Omron CX-Programmer project 新工程 (CX-Programmer 9.73)

# PLC 新PLC1: C200HE CPU42

## Program 新程序1 (no task)
; [项目]：本项目是为“台湾大拉无板”自动化拉丝生产线设计的控制系统，通过PLC实现生产线的自动化管理。系统包含启动、错误处理、定时管理、事件计数和设备驱动模块，确保拉丝作业的正常运行。 / [设备信息]：系统涉及的物理设备包括启动按钮、停止按钮、模式选择按钮、传感器、拉丝机电机和阀门。 / [系统执行]：系统通过启动按钮启动生产线，操作员按下按钮后，程序检查异常传感器1至10是否正常。 / 若无异常且延时定时器2未超时，置位运行模式标志，此时生产线进入运行状态。 / 特别地，运行模式标志只有在启动按钮按下后才会置位，避免未触发启动时生产线意外运行。 / 运行时，电机控制1至10驱动拉丝机运转，其中电机控制1的激活必须在运行模式标志置位时才能发生，防止模式未启用时设备误动作。 / 当系统正常运行时，若检测到特定条件，激活电机控制1以驱动设备。 / 启动时，异常传感器1至10检查是否正常；运行中，若任一传感器检测到异常，则置位相应标志。 / 若延时定时器1超时，置位错误状态标志；随后通过停止控制信号停止生产线，并激活阀门2发出警报。 / 错误状态标志置位后，激活阀门2发出警报，并通过停止控制信号停止生产线。 / 延时定时器1超时置位错误状态标志；延时定时器2超时（设定为20个时间单位）后，也触发类似逻辑。 / 操作员可通过手动按钮1和手动按钮2手动控制阀门1和阀门2（如调节润滑液或冷却液），这些操作的计数记录在次数记录区中。 / 当计数达到4时，系统自动复位阀门状态，确保手动操作不会无限制累积。 / 事件计数器1记录拉丝次数，限值为3次；若达到限值，后续逻辑触发警报。 / 模式选择按钮1至9允许切换拉丝模式（如高速或低速模式），当前模式存储在模式记录区中，影响拉丝参数。 / 参数存储区保存运行数据和历史记录，便于维护和故障排查。 / 按下停止按钮后，系统置位停止控制信号以停止生产线。

### Section 段1

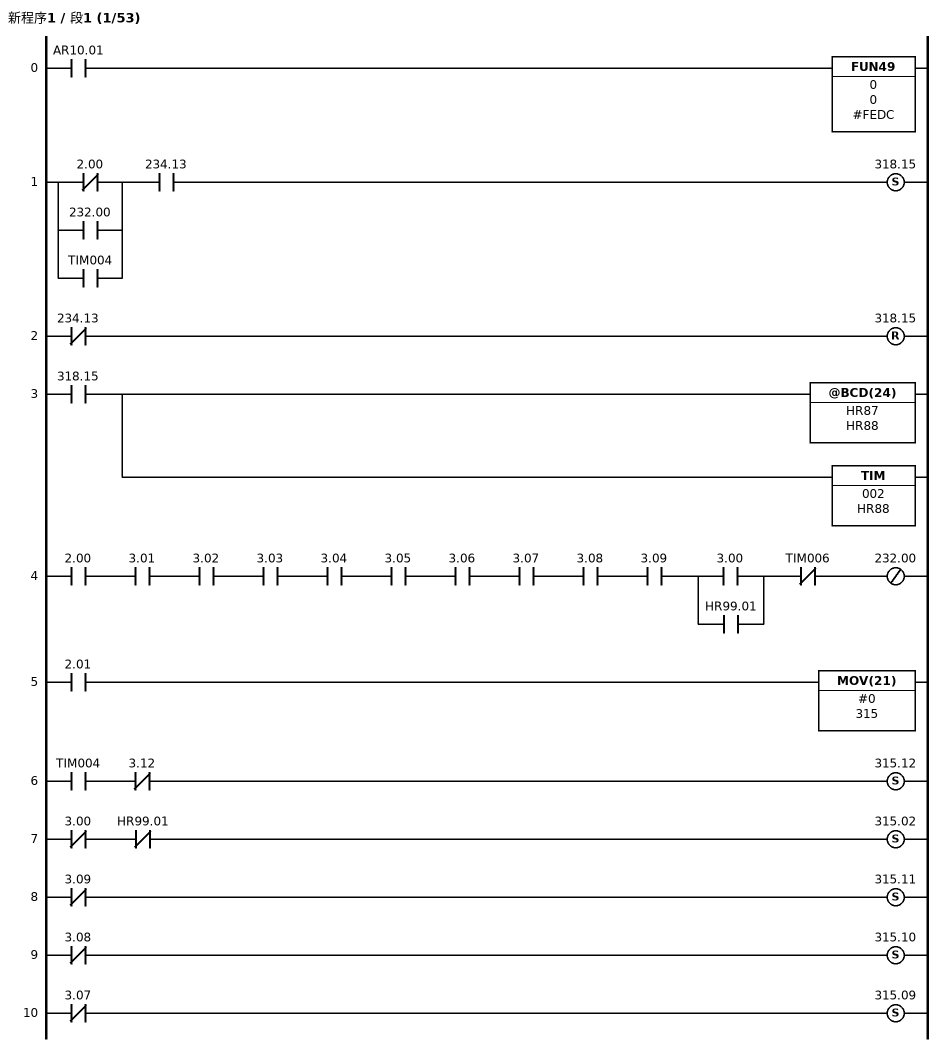
; rung 0
LD AR10.01
FUN49 0 0 #FEDC
; rung 1
LDNOT 2.00
OR 232.00
OR TIM004
AND 234.13
SET 318.15
; rung 2
LDNOT 234.13
RSET 318.15
; rung 3
LD 318.15
@BCD(24) HR87 HR88
TIM 002 HR88
; rung 4
LD 2.00
AND 3.01
AND 3.02
AND 3.03
AND 3.04
AND 3.05
AND 3.06
AND 3.07
AND 3.08
AND 3.09
LD 3.00
OR HR99.01
ANDLD
ANDNOT TIM006
OUTNOT 232.00
; rung 5
LD 2.01
MOV(21) #0 315
; rung 6
LD TIM004
ANDNOT 3.12
SET 315.12
; rung 7
LDNOT 3.00
ANDNOT HR99.01
SET 315.02
; rung 8
LDNOT 3.09
SET 315.11
; rung 9
LDNOT 3.08
SET 315.10
; rung 10
LDNOT 3.07
SET 315.09

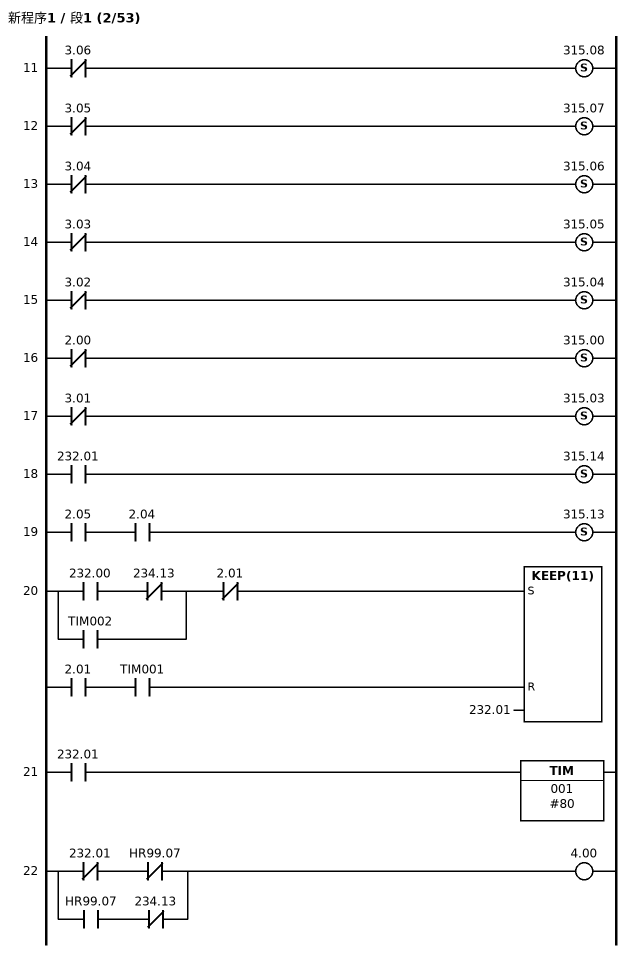
; rung 11
LDNOT 3.06
SET 315.08
; rung 12
LDNOT 3.05
SET 315.07
; rung 13
LDNOT 3.04
SET 315.06
; rung 14
LDNOT 3.03
SET 315.05
; rung 15
LDNOT 3.02
SET 315.04
; rung 16
LDNOT 2.00
SET 315.00
; rung 17
LDNOT 3.01
SET 315.03
; rung 18
LD 232.01
SET 315.14
; rung 19
LD 2.05
AND 2.04
SET 315.13
; rung 20
LD 232.00
ANDNOT 234.13
OR TIM002
ANDNOT 2.01
LD 2.01
AND TIM001
KEEP(11) 232.01
; rung 21
LD 232.01
TIM 001 #80
; rung 22
LDNOT 232.01
ANDNOT HR99.07
LD HR99.07
ANDNOT 234.13
ORLD
OUT 4.00

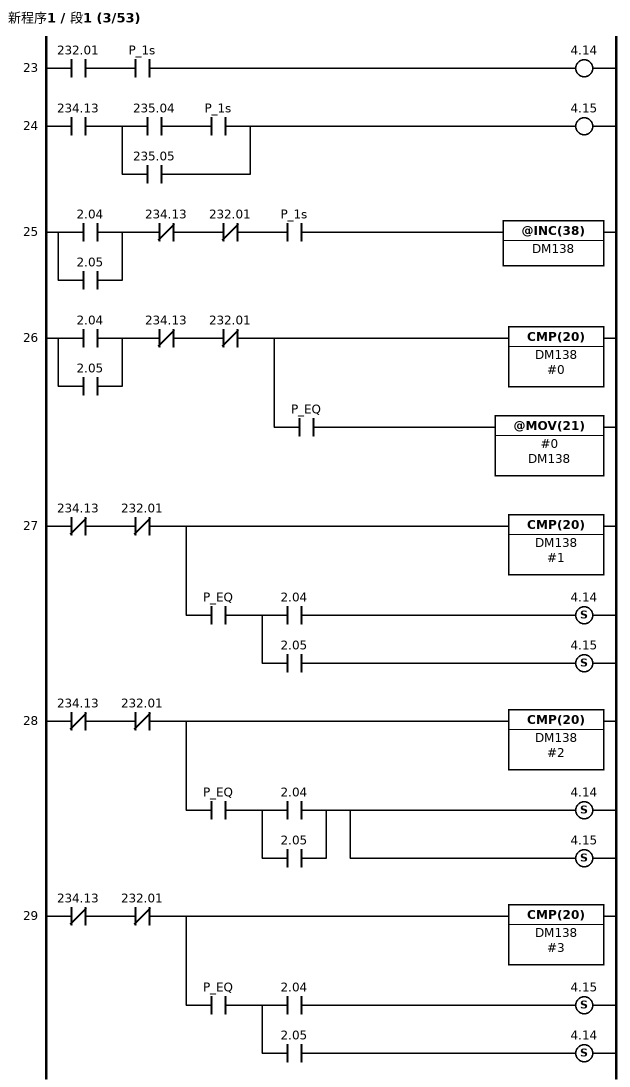
; rung 23
LD 232.01
AND P_1s
OUT 4.14
; rung 24
LD 234.13
LD 235.04
AND P_1s
OR 235.05
ANDLD
OUT 4.15
; rung 25
LD 2.04
OR 2.05
ANDNOT 234.13
ANDNOT 232.01
AND P_1s
@INC(38) DM138
; rung 26
LD 2.04
OR 2.05
ANDNOT 234.13
ANDNOT 232.01
CMP(20) DM138 #0
AND P_EQ
@MOV(21) #0 DM138
; rung 27
LDNOT 234.13
ANDNOT 232.01
CMP(20) DM138 #1
AND P_EQ
OUT TR0
AND 2.04
SET 4.14
LD TR0
AND 2.05
SET 4.15
; rung 28
LDNOT 234.13
ANDNOT 232.01
CMP(20) DM138 #2
AND P_EQ
LD 2.04
OR 2.05
ANDLD
SET 4.14
SET 4.15
; rung 29
LDNOT 234.13
ANDNOT 232.01
CMP(20) DM138 #3
AND P_EQ
OUT TR0
AND 2.04
SET 4.15
LD TR0
AND 2.05
SET 4.14

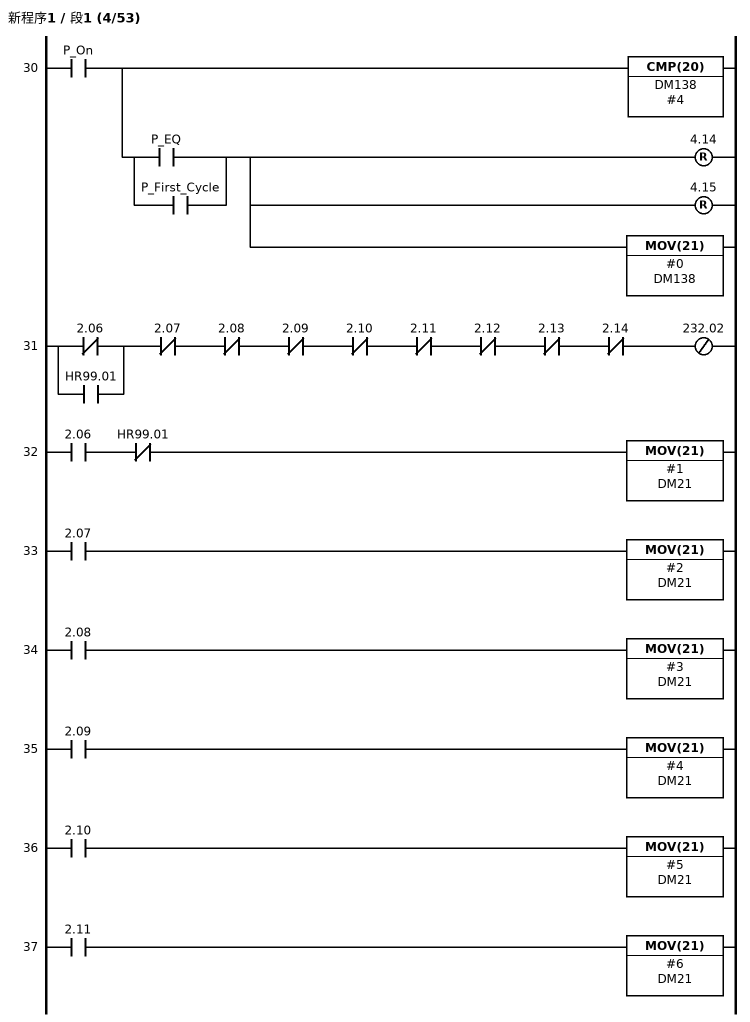
; rung 30
LD P_On
CMP(20) DM138 #4
LD P_EQ
OR P_First_Cycle
ANDLD
RSET 4.14
RSET 4.15
MOV(21) #0 DM138
; rung 31
LDNOT 2.06
OR HR99.01
ANDNOT 2.07
ANDNOT 2.08
ANDNOT 2.09
ANDNOT 2.10
ANDNOT 2.11
ANDNOT 2.12
ANDNOT 2.13
ANDNOT 2.14
OUTNOT 232.02
; rung 32
LD 2.06
ANDNOT HR99.01
MOV(21) #1 DM21
; rung 33
LD 2.07
MOV(21) #2 DM21
; rung 34
LD 2.08
MOV(21) #3 DM21
; rung 35
LD 2.09
MOV(21) #4 DM21
; rung 36
LD 2.10
MOV(21) #5 DM21
; rung 37
LD 2.11
MOV(21) #6 DM21

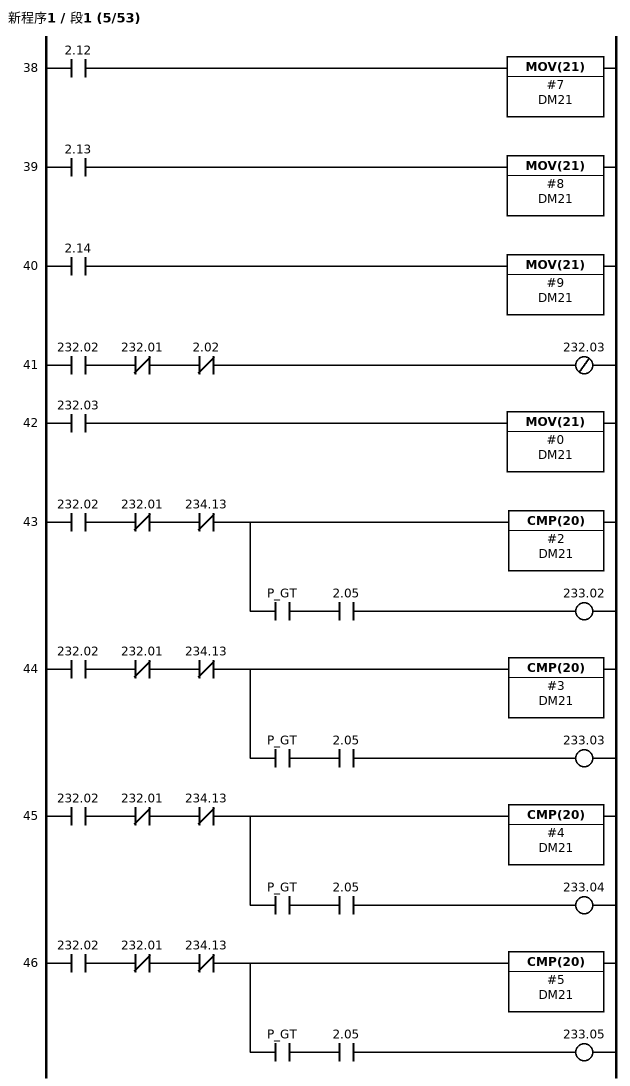
; rung 38
LD 2.12
MOV(21) #7 DM21
; rung 39
LD 2.13
MOV(21) #8 DM21
; rung 40
LD 2.14
MOV(21) #9 DM21
; rung 41
LD 232.02
ANDNOT 232.01
ANDNOT 2.02
OUTNOT 232.03
; rung 42
LD 232.03
MOV(21) #0 DM21
; rung 43
LD 232.02
ANDNOT 232.01
ANDNOT 234.13
CMP(20) #2 DM21
AND P_GT
AND 2.05
OUT 233.02
; rung 44
LD 232.02
ANDNOT 232.01
ANDNOT 234.13
CMP(20) #3 DM21
AND P_GT
AND 2.05
OUT 233.03
; rung 45
LD 232.02
ANDNOT 232.01
ANDNOT 234.13
CMP(20) #4 DM21
AND P_GT
AND 2.05
OUT 233.04
; rung 46
LD 232.02
ANDNOT 232.01
ANDNOT 234.13
CMP(20) #5 DM21
AND P_GT
AND 2.05
OUT 233.05

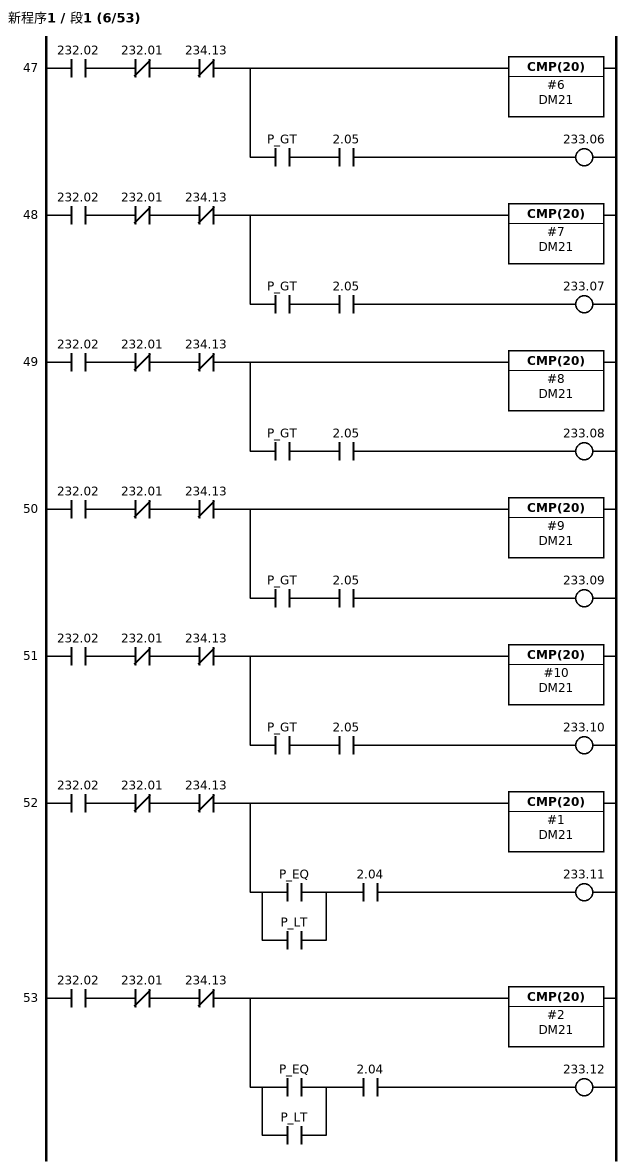
; rung 47
LD 232.02
ANDNOT 232.01
ANDNOT 234.13
CMP(20) #6 DM21
AND P_GT
AND 2.05
OUT 233.06
; rung 48
LD 232.02
ANDNOT 232.01
ANDNOT 234.13
CMP(20) #7 DM21
AND P_GT
AND 2.05
OUT 233.07
; rung 49
LD 232.02
ANDNOT 232.01
ANDNOT 234.13
CMP(20) #8 DM21
AND P_GT
AND 2.05
OUT 233.08
; rung 50
LD 232.02
ANDNOT 232.01
ANDNOT 234.13
CMP(20) #9 DM21
AND P_GT
AND 2.05
OUT 233.09
; rung 51
LD 232.02
ANDNOT 232.01
ANDNOT 234.13
CMP(20) #10 DM21
AND P_GT
AND 2.05
OUT 233.10
; rung 52
LD 232.02
ANDNOT 232.01
ANDNOT 234.13
CMP(20) #1 DM21
LD P_EQ
OR P_LT
AND 2.04
ANDLD
OUT 233.11
; rung 53
LD 232.02
ANDNOT 232.01
ANDNOT 234.13
CMP(20) #2 DM21
LD P_EQ
OR P_LT
AND 2.04
ANDLD
OUT 233.12

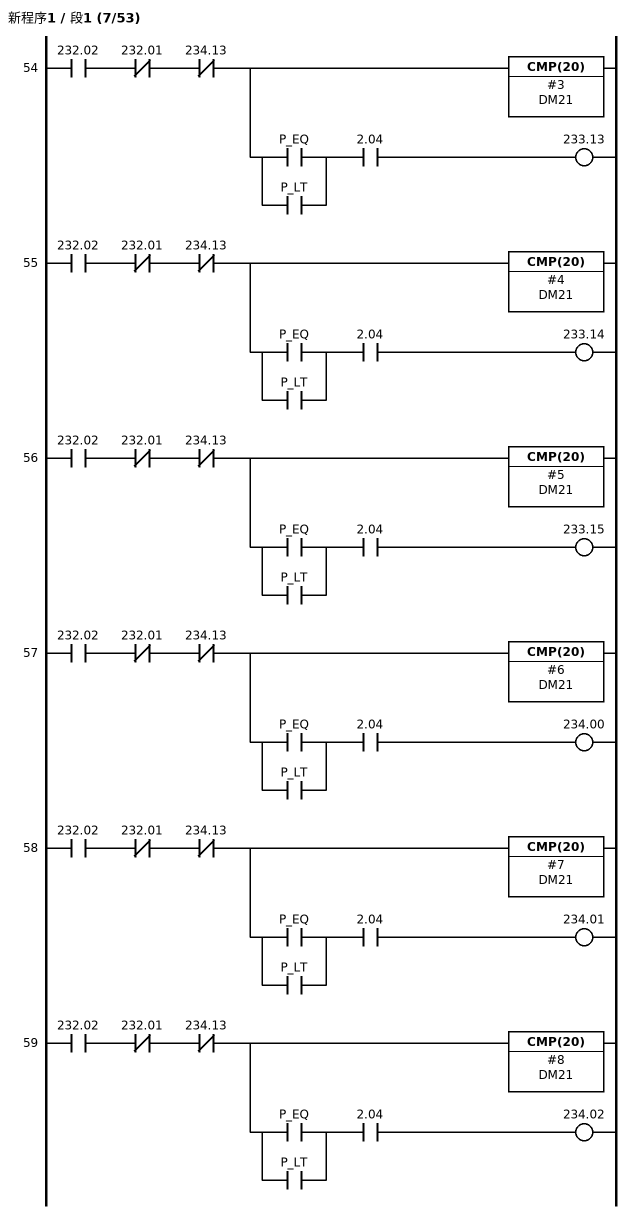
; rung 54
LD 232.02
ANDNOT 232.01
ANDNOT 234.13
CMP(20) #3 DM21
LD P_EQ
OR P_LT
AND 2.04
ANDLD
OUT 233.13
; rung 55
LD 232.02
ANDNOT 232.01
ANDNOT 234.13
CMP(20) #4 DM21
LD P_EQ
OR P_LT
AND 2.04
ANDLD
OUT 233.14
; rung 56
LD 232.02
ANDNOT 232.01
ANDNOT 234.13
CMP(20) #5 DM21
LD P_EQ
OR P_LT
AND 2.04
ANDLD
OUT 233.15
; rung 57
LD 232.02
ANDNOT 232.01
ANDNOT 234.13
CMP(20) #6 DM21
LD P_EQ
OR P_LT
AND 2.04
ANDLD
OUT 234.00
; rung 58
LD 232.02
ANDNOT 232.01
ANDNOT 234.13
CMP(20) #7 DM21
LD P_EQ
OR P_LT
AND 2.04
ANDLD
OUT 234.01
; rung 59
LD 232.02
ANDNOT 232.01
ANDNOT 234.13
CMP(20) #8 DM21
LD P_EQ
OR P_LT
AND 2.04
ANDLD
OUT 234.02

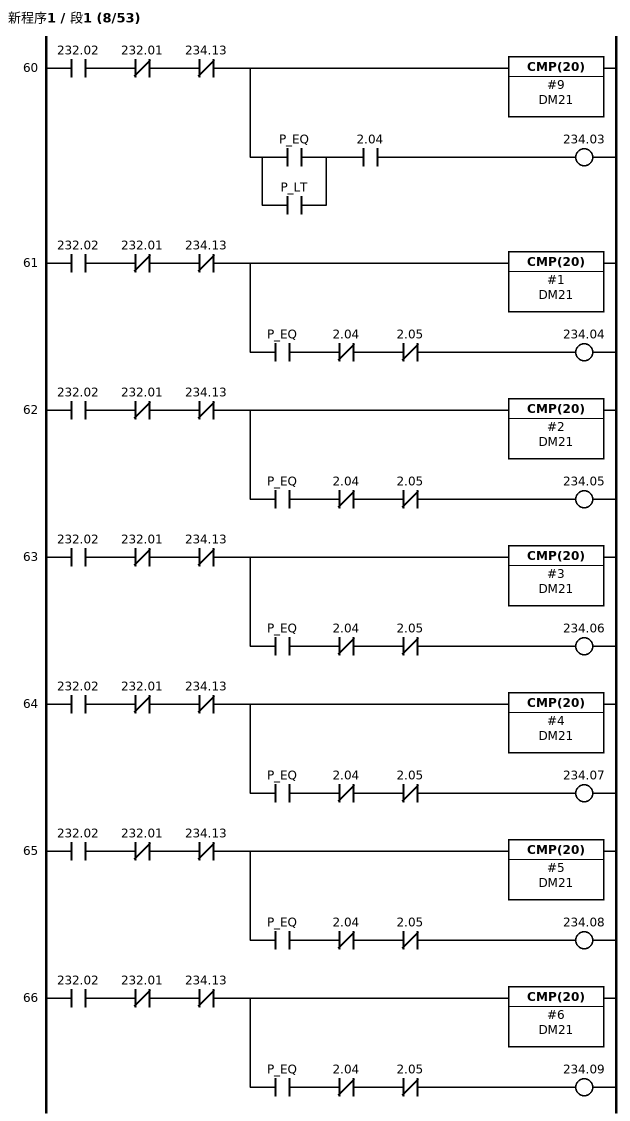
; rung 60
LD 232.02
ANDNOT 232.01
ANDNOT 234.13
CMP(20) #9 DM21
LD P_EQ
OR P_LT
AND 2.04
ANDLD
OUT 234.03
; rung 61
LD 232.02
ANDNOT 232.01
ANDNOT 234.13
CMP(20) #1 DM21
AND P_EQ
ANDNOT 2.04
ANDNOT 2.05
OUT 234.04
; rung 62
LD 232.02
ANDNOT 232.01
ANDNOT 234.13
CMP(20) #2 DM21
AND P_EQ
ANDNOT 2.04
ANDNOT 2.05
OUT 234.05
; rung 63
LD 232.02
ANDNOT 232.01
ANDNOT 234.13
CMP(20) #3 DM21
AND P_EQ
ANDNOT 2.04
ANDNOT 2.05
OUT 234.06
; rung 64
LD 232.02
ANDNOT 232.01
ANDNOT 234.13
CMP(20) #4 DM21
AND P_EQ
ANDNOT 2.04
ANDNOT 2.05
OUT 234.07
; rung 65
LD 232.02
ANDNOT 232.01
ANDNOT 234.13
CMP(20) #5 DM21
AND P_EQ
ANDNOT 2.04
ANDNOT 2.05
OUT 234.08
; rung 66
LD 232.02
ANDNOT 232.01
ANDNOT 234.13
CMP(20) #6 DM21
AND P_EQ
ANDNOT 2.04
ANDNOT 2.05
OUT 234.09

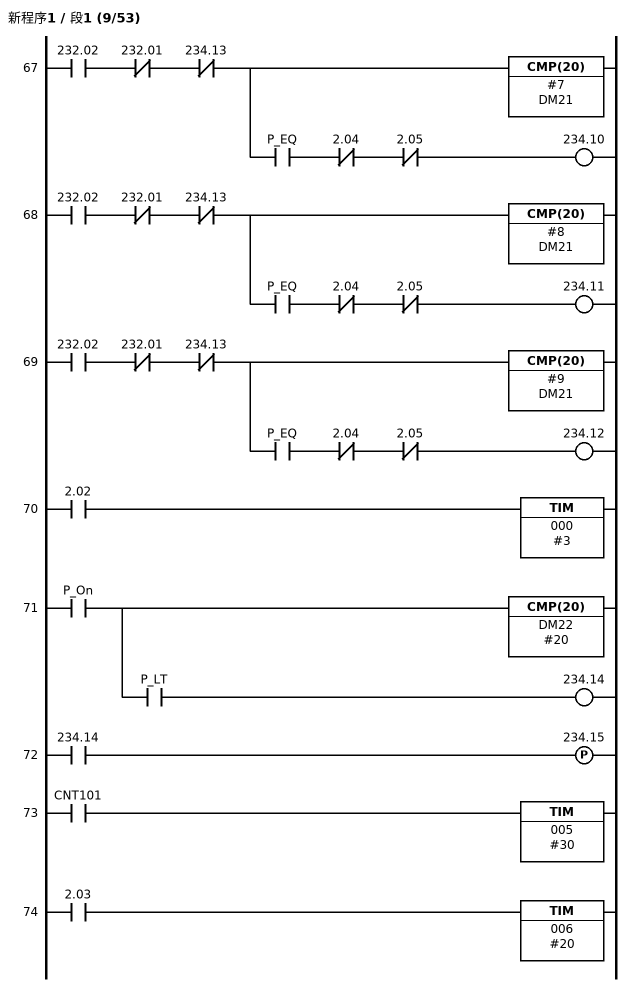
; rung 67
LD 232.02
ANDNOT 232.01
ANDNOT 234.13
CMP(20) #7 DM21
AND P_EQ
ANDNOT 2.04
ANDNOT 2.05
OUT 234.10
; rung 68
LD 232.02
ANDNOT 232.01
ANDNOT 234.13
CMP(20) #8 DM21
AND P_EQ
ANDNOT 2.04
ANDNOT 2.05
OUT 234.11
; rung 69
LD 232.02
ANDNOT 232.01
ANDNOT 234.13
CMP(20) #9 DM21
AND P_EQ
ANDNOT 2.04
ANDNOT 2.05
OUT 234.12
; rung 70
LD 2.02
TIM 000 #3
; rung 71
LD P_On
CMP(20) DM22 #20
AND P_LT
OUT 234.14
; rung 72
LD 234.14
DIFU(13) 234.15
; rung 73
LD CNT101
TIM 005 #30
; rung 74
LD 2.03
TIM 006 #20

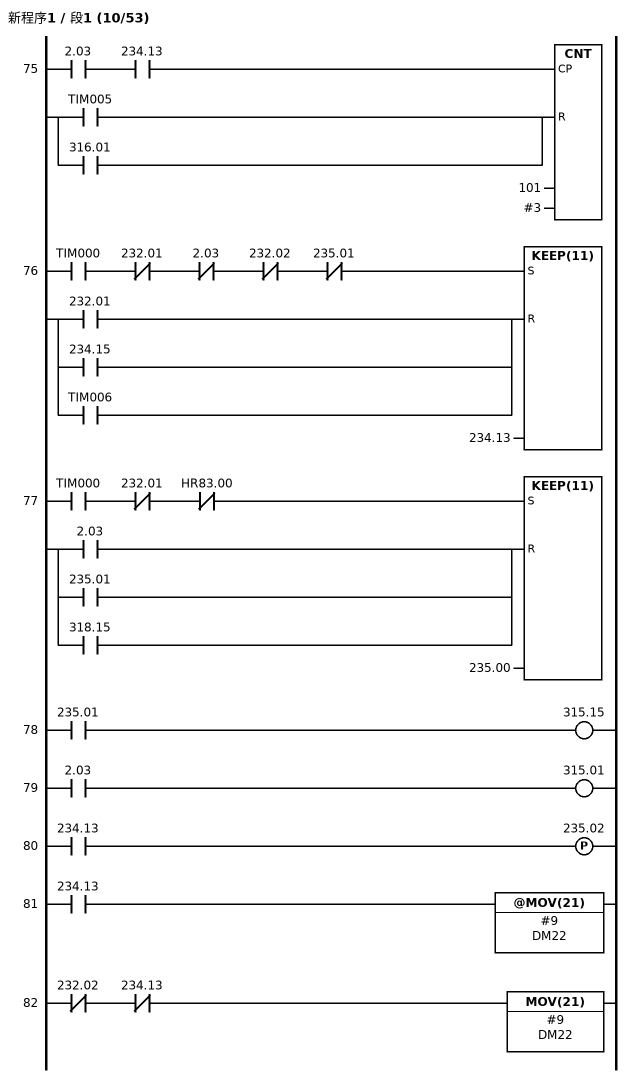
; rung 75
LD 2.03
AND 234.13
LD TIM005
OR 316.01
CNT 101 #3
; rung 76
LD TIM000
ANDNOT 232.01
ANDNOT 2.03
ANDNOT 232.02
ANDNOT 235.01
LD 232.01
OR 234.15
OR TIM006
KEEP(11) 234.13
; rung 77
LD TIM000
ANDNOT 232.01
ANDNOT HR83.00
LD 2.03
OR 235.01
OR 318.15
KEEP(11) 235.00
; rung 78
LD 235.01
OUT 315.15
; rung 79
LD 2.03
OUT 315.01
; rung 80
LD 234.13
DIFU(13) 235.02
; rung 81
LD 234.13
@MOV(21) #9 DM22
; rung 82
LDNOT 232.02
ANDNOT 234.13
MOV(21) #9 DM22

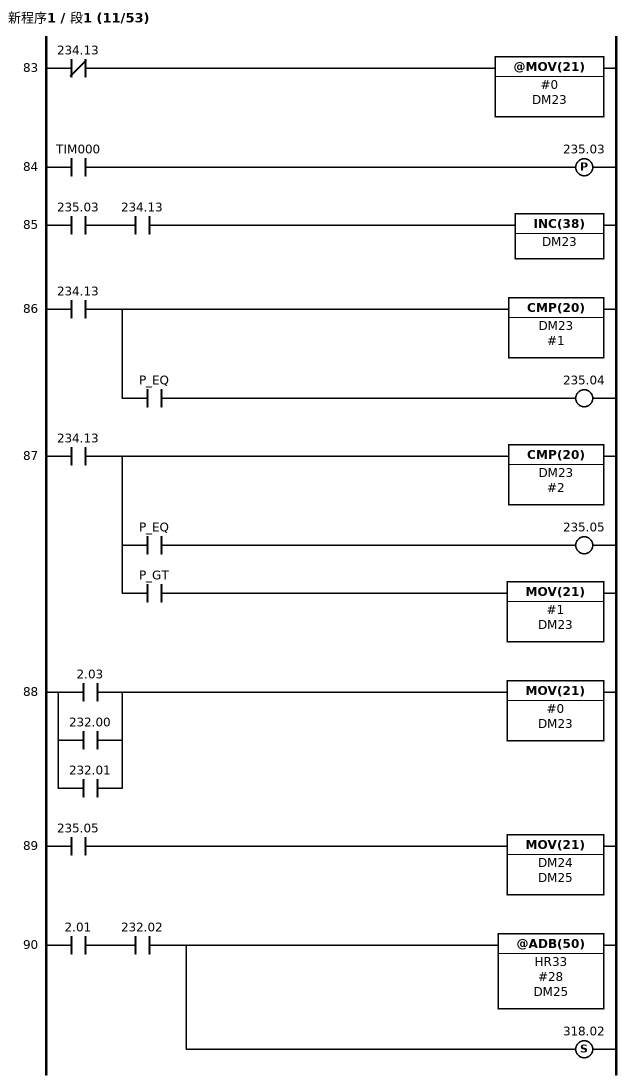
; rung 83
LDNOT 234.13
@MOV(21) #0 DM23
; rung 84
LD TIM000
DIFU(13) 235.03
; rung 85
LD 235.03
AND 234.13
INC(38) DM23
; rung 86
LD 234.13
CMP(20) DM23 #1
AND P_EQ
OUT 235.04
; rung 87
LD 234.13
OUT TR0
CMP(20) DM23 #2
AND P_EQ
OUT 235.05
LD TR0
AND P_GT
MOV(21) #1 DM23
; rung 88
LD 2.03
OR 232.00
OR 232.01
MOV(21) #0 DM23
; rung 89
LD 235.05
MOV(21) DM24 DM25
; rung 90
LD 2.01
AND 232.02
@ADB(50) HR33 #28 DM25
SET 318.02

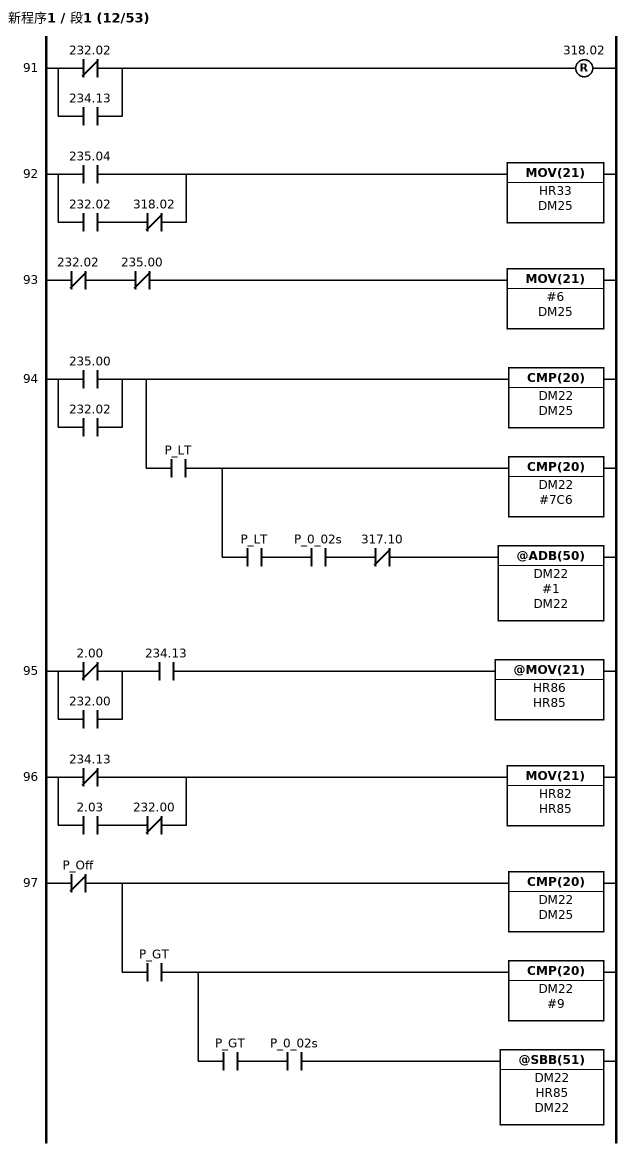
; rung 91
LDNOT 232.02
OR 234.13
RSET 318.02
; rung 92
LD 235.04
LD 232.02
ANDNOT 318.02
ORLD
MOV(21) HR33 DM25
; rung 93
LDNOT 232.02
ANDNOT 235.00
MOV(21) #6 DM25
; rung 94
LD 235.00
OR 232.02
CMP(20) DM22 DM25
AND P_LT
CMP(20) DM22 #7C6
AND P_LT
AND P_0_02s
ANDNOT 317.10
@ADB(50) DM22 #1 DM22
; rung 95
LDNOT 2.00
OR 232.00
AND 234.13
@MOV(21) HR86 HR85
; rung 96
LDNOT 234.13
LD 2.03
ANDNOT 232.00
ORLD
MOV(21) HR82 HR85
; rung 97
LDNOT P_Off
CMP(20) DM22 DM25
AND P_GT
CMP(20) DM22 #9
AND P_GT
AND P_0_02s
@SBB(51) DM22 HR85 DM22

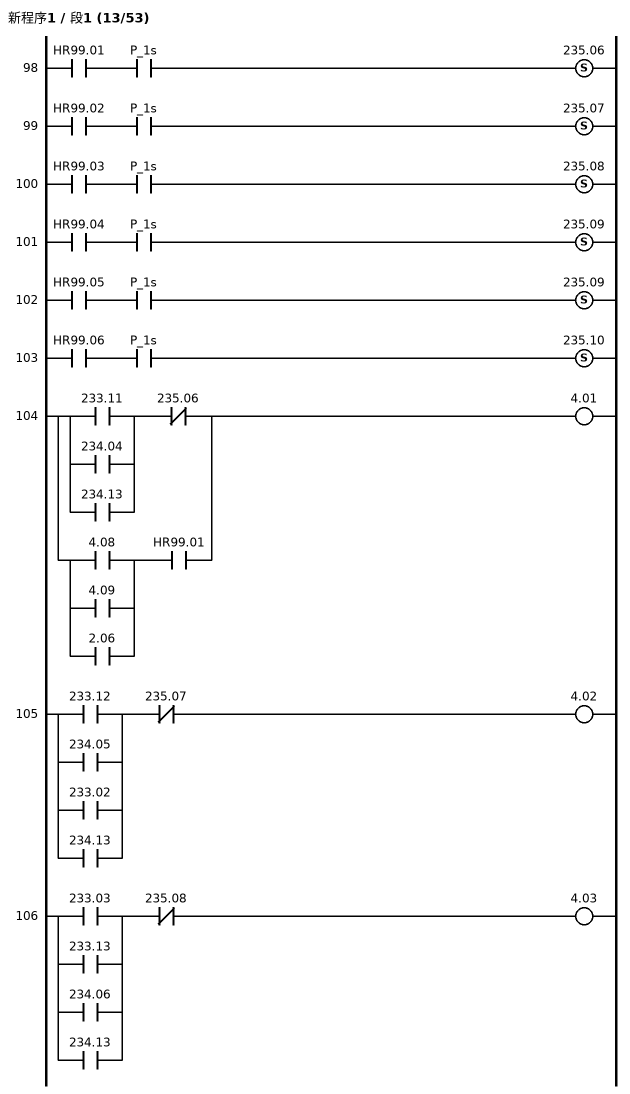
; rung 98
LD HR99.01
AND P_1s
SET 235.06
; rung 99
LD HR99.02
AND P_1s
SET 235.07
; rung 100
LD HR99.03
AND P_1s
SET 235.08
; rung 101
LD HR99.04
AND P_1s
SET 235.09
; rung 102
LD HR99.05
AND P_1s
SET 235.09
; rung 103
LD HR99.06
AND P_1s
SET 235.10
; rung 104
LD 233.11
OR 234.04
OR 234.13
ANDNOT 235.06
LD 4.08
OR 4.09
OR 2.06
AND HR99.01
ORLD
OUT 4.01
; rung 105
LD 233.12
OR 234.05
OR 233.02
OR 234.13
ANDNOT 235.07
OUT 4.02
; rung 106
LD 233.03
OR 233.13
OR 234.06
OR 234.13
ANDNOT 235.08
OUT 4.03

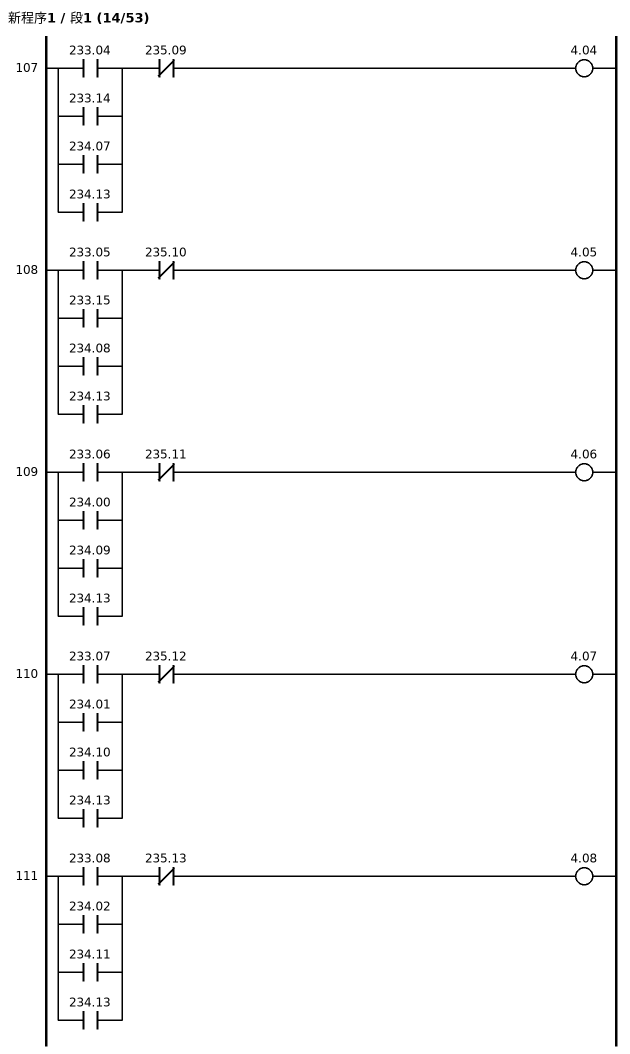
; rung 107
LD 233.04
OR 233.14
OR 234.07
OR 234.13
ANDNOT 235.09
OUT 4.04
; rung 108
LD 233.05
OR 233.15
OR 234.08
OR 234.13
ANDNOT 235.10
OUT 4.05
; rung 109
LD 233.06
OR 234.00
OR 234.09
OR 234.13
ANDNOT 235.11
OUT 4.06
; rung 110
LD 233.07
OR 234.01
OR 234.10
OR 234.13
ANDNOT 235.12
OUT 4.07
; rung 111
LD 233.08
OR 234.02
OR 234.11
OR 234.13
ANDNOT 235.13
OUT 4.08

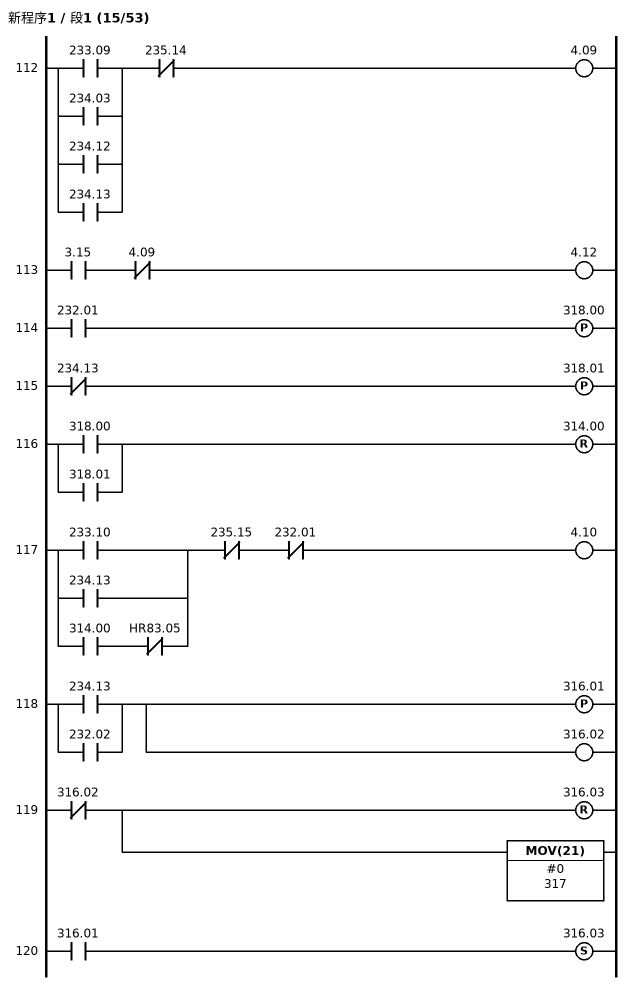
; rung 112
LD 233.09
OR 234.03
OR 234.12
OR 234.13
ANDNOT 235.14
OUT 4.09
; rung 113
LD 3.15
ANDNOT 4.09
OUT 4.12
; rung 114
LD 232.01
DIFU(13) 318.00
; rung 115
LDNOT 234.13
DIFU(13) 318.01
; rung 116
LD 318.00
OR 318.01
RSET 314.00
; rung 117
LD 233.10
OR 234.13
LD 314.00
ANDNOT HR83.05
ORLD
ANDNOT 235.15
ANDNOT 232.01
OUT 4.10
; rung 118
LD 234.13
OR 232.02
DIFU(13) 316.01
OUT 316.02
; rung 119
LDNOT 316.02
RSET 316.03
MOV(21) #0 317
; rung 120
LD 316.01
SET 316.03

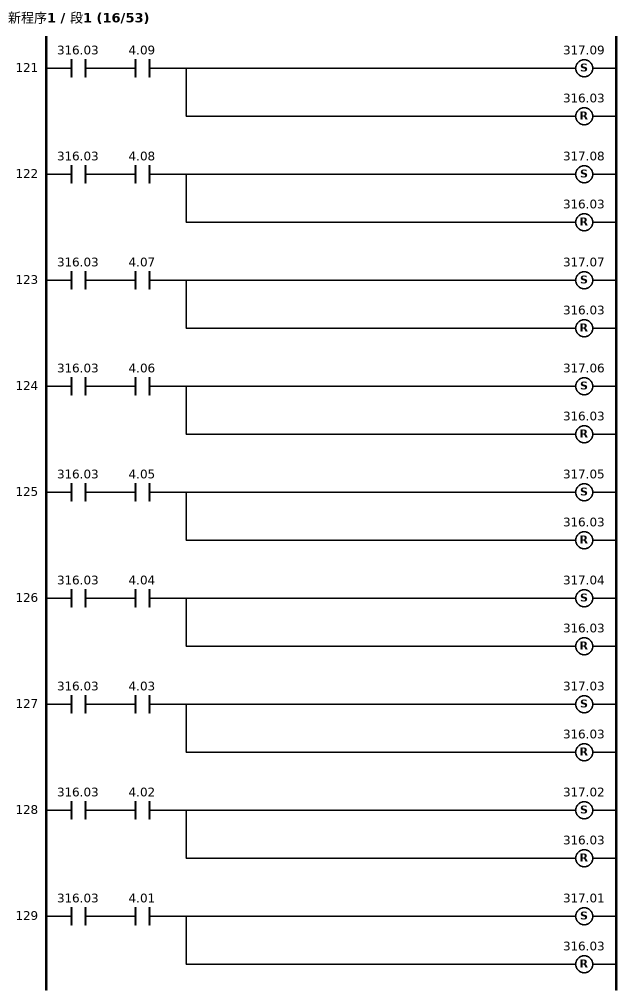
; rung 121
LD 316.03
AND 4.09
SET 317.09
RSET 316.03
; rung 122
LD 316.03
AND 4.08
SET 317.08
RSET 316.03
; rung 123
LD 316.03
AND 4.07
SET 317.07
RSET 316.03
; rung 124
LD 316.03
AND 4.06
SET 317.06
RSET 316.03
; rung 125
LD 316.03
AND 4.05
SET 317.05
RSET 316.03
; rung 126
LD 316.03
AND 4.04
SET 317.04
RSET 316.03
; rung 127
LD 316.03
AND 4.03
SET 317.03
RSET 316.03
; rung 128
LD 316.03
AND 4.02
SET 317.02
RSET 316.03
; rung 129
LD 316.03
AND 4.01
SET 317.01
RSET 316.03

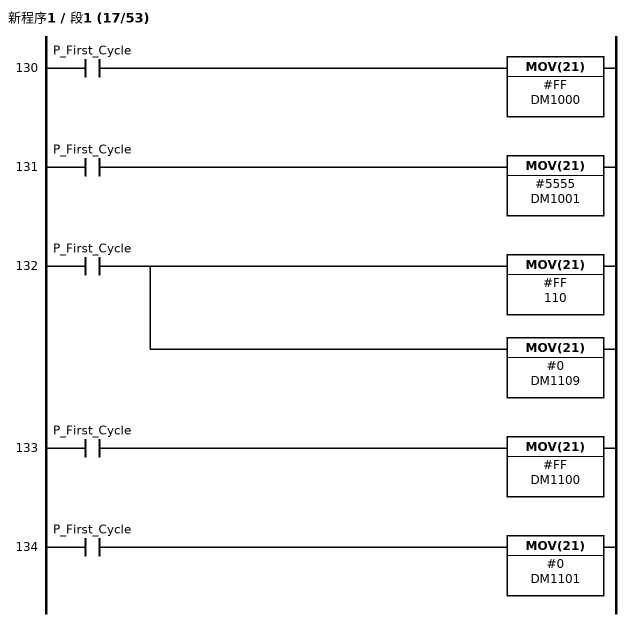
; rung 130
LD P_First_Cycle
MOV(21) #FF DM1000
; rung 131
LD P_First_Cycle
MOV(21) #5555 DM1001
; rung 132
LD P_First_Cycle
MOV(21) #FF 110
MOV(21) #0 DM1109
; rung 133
LD P_First_Cycle
MOV(21) #FF DM1100
; rung 134
LD P_First_Cycle
MOV(21) #0 DM1101

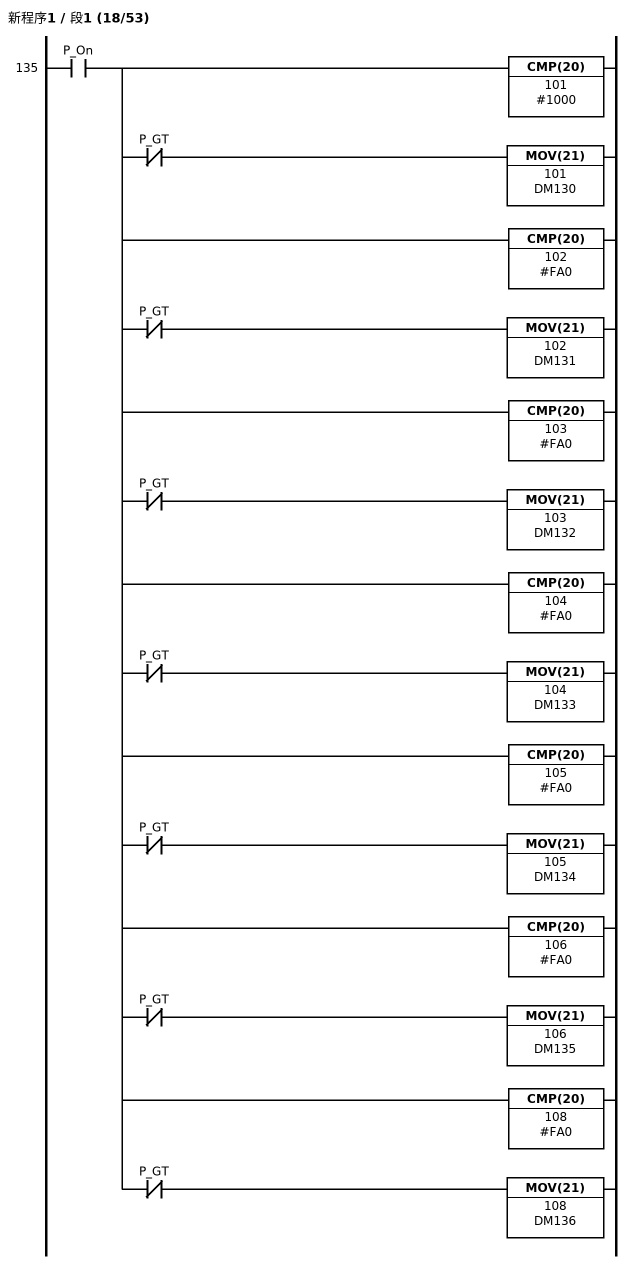
; rung 135
LD P_On
OUT TR0
CMP(20) 101 #1000
ANDNOT P_GT
MOV(21) 101 DM130
LD TR0
CMP(20) 102 #FA0
ANDNOT P_GT
MOV(21) 102 DM131
LD TR0
CMP(20) 103 #FA0
ANDNOT P_GT
MOV(21) 103 DM132
LD TR0
CMP(20) 104 #FA0
ANDNOT P_GT
MOV(21) 104 DM133
LD TR0
CMP(20) 105 #FA0
ANDNOT P_GT
MOV(21) 105 DM134
LD TR0
CMP(20) 106 #FA0
ANDNOT P_GT
MOV(21) 106 DM135
LD TR0
CMP(20) 108 #FA0
ANDNOT P_GT
MOV(21) 108 DM136

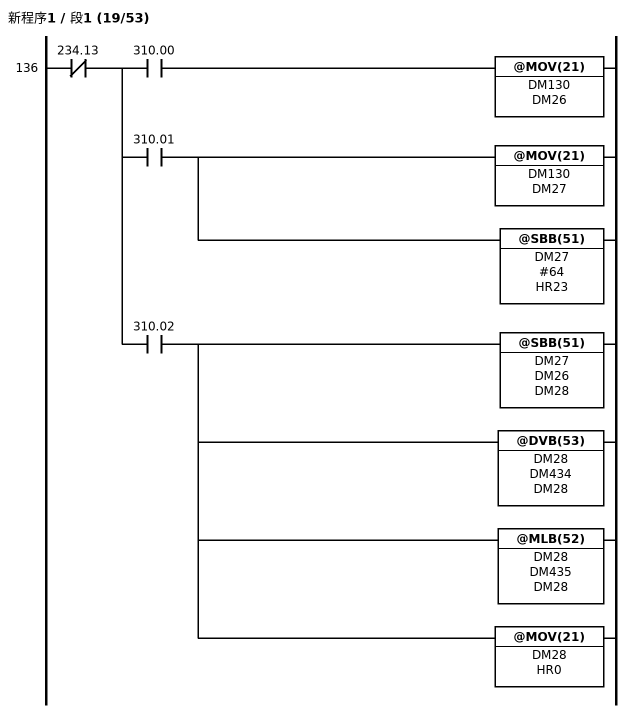
; rung 136
LDNOT 234.13
OUT TR0
AND 310.00
@MOV(21) DM130 DM26
LD TR0
AND 310.01
@MOV(21) DM130 DM27
@SBB(51) DM27 #64 HR23
LD TR0
AND 310.02
@SBB(51) DM27 DM26 DM28
@DVB(53) DM28 DM434 DM28
@MLB(52) DM28 DM435 DM28
@MOV(21) DM28 HR0

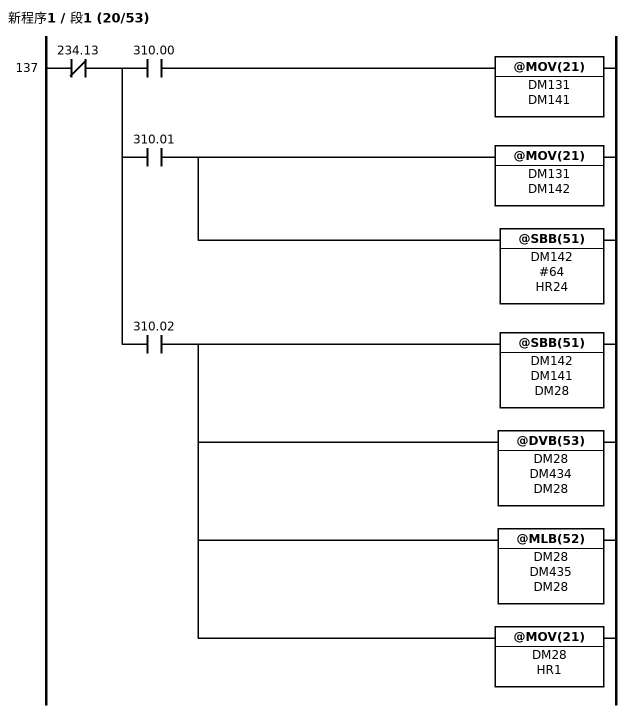
; rung 137
LDNOT 234.13
OUT TR0
AND 310.00
@MOV(21) DM131 DM141
LD TR0
AND 310.01
@MOV(21) DM131 DM142
@SBB(51) DM142 #64 HR24
LD TR0
AND 310.02
@SBB(51) DM142 DM141 DM28
@DVB(53) DM28 DM434 DM28
@MLB(52) DM28 DM435 DM28
@MOV(21) DM28 HR1

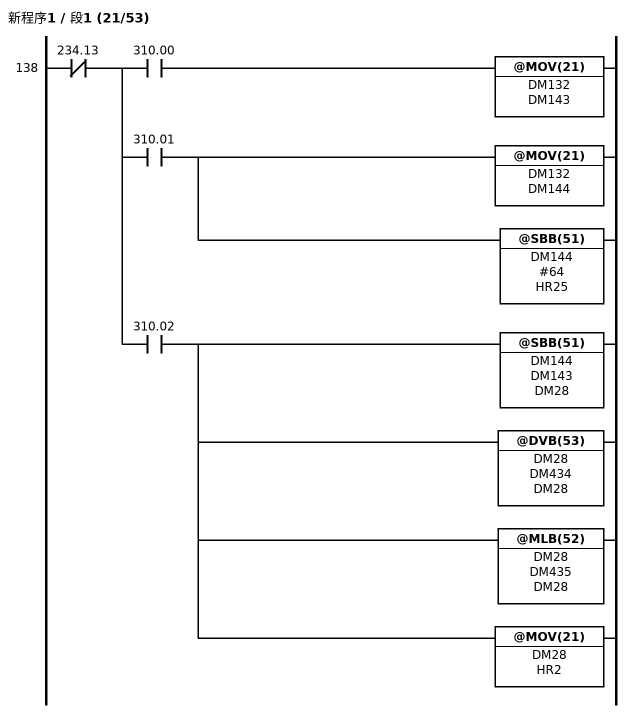
; rung 138
LDNOT 234.13
OUT TR0
AND 310.00
@MOV(21) DM132 DM143
LD TR0
AND 310.01
@MOV(21) DM132 DM144
@SBB(51) DM144 #64 HR25
LD TR0
AND 310.02
@SBB(51) DM144 DM143 DM28
@DVB(53) DM28 DM434 DM28
@MLB(52) DM28 DM435 DM28
@MOV(21) DM28 HR2

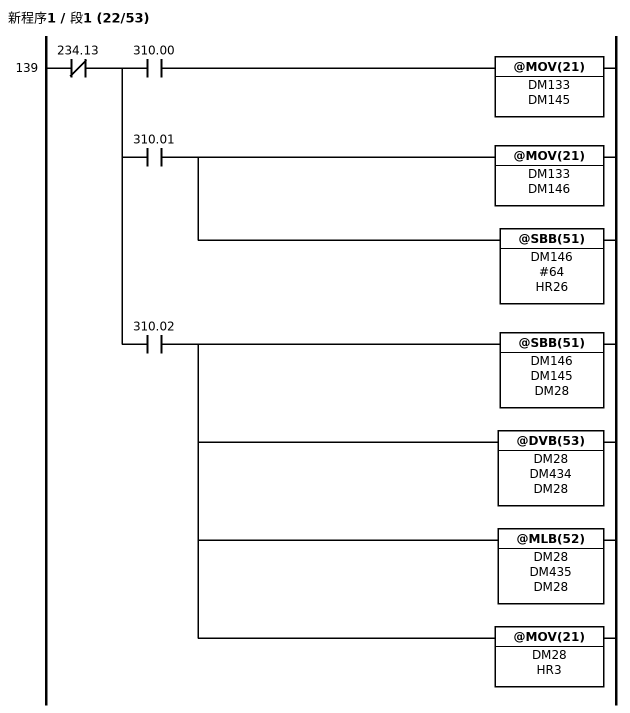
; rung 139
LDNOT 234.13
OUT TR0
AND 310.00
@MOV(21) DM133 DM145
LD TR0
AND 310.01
@MOV(21) DM133 DM146
@SBB(51) DM146 #64 HR26
LD TR0
AND 310.02
@SBB(51) DM146 DM145 DM28
@DVB(53) DM28 DM434 DM28
@MLB(52) DM28 DM435 DM28
@MOV(21) DM28 HR3

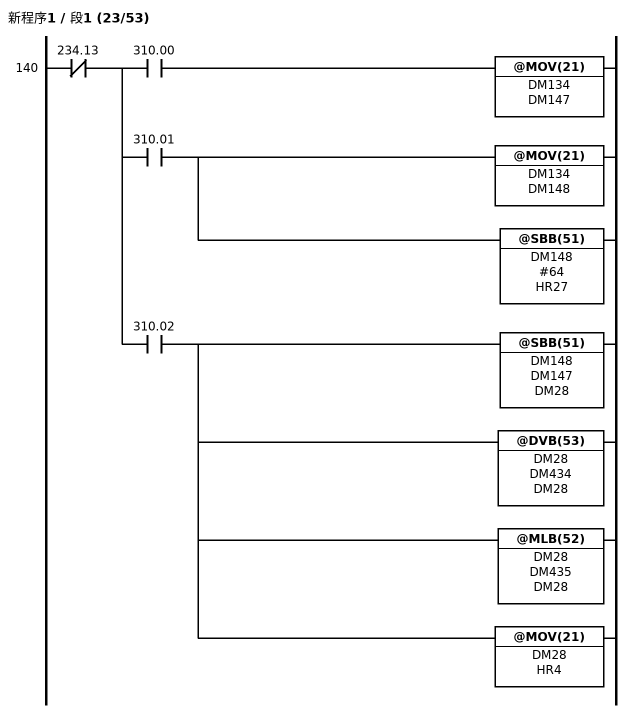
; rung 140
LDNOT 234.13
OUT TR0
AND 310.00
@MOV(21) DM134 DM147
LD TR0
AND 310.01
@MOV(21) DM134 DM148
@SBB(51) DM148 #64 HR27
LD TR0
AND 310.02
@SBB(51) DM148 DM147 DM28
@DVB(53) DM28 DM434 DM28
@MLB(52) DM28 DM435 DM28
@MOV(21) DM28 HR4

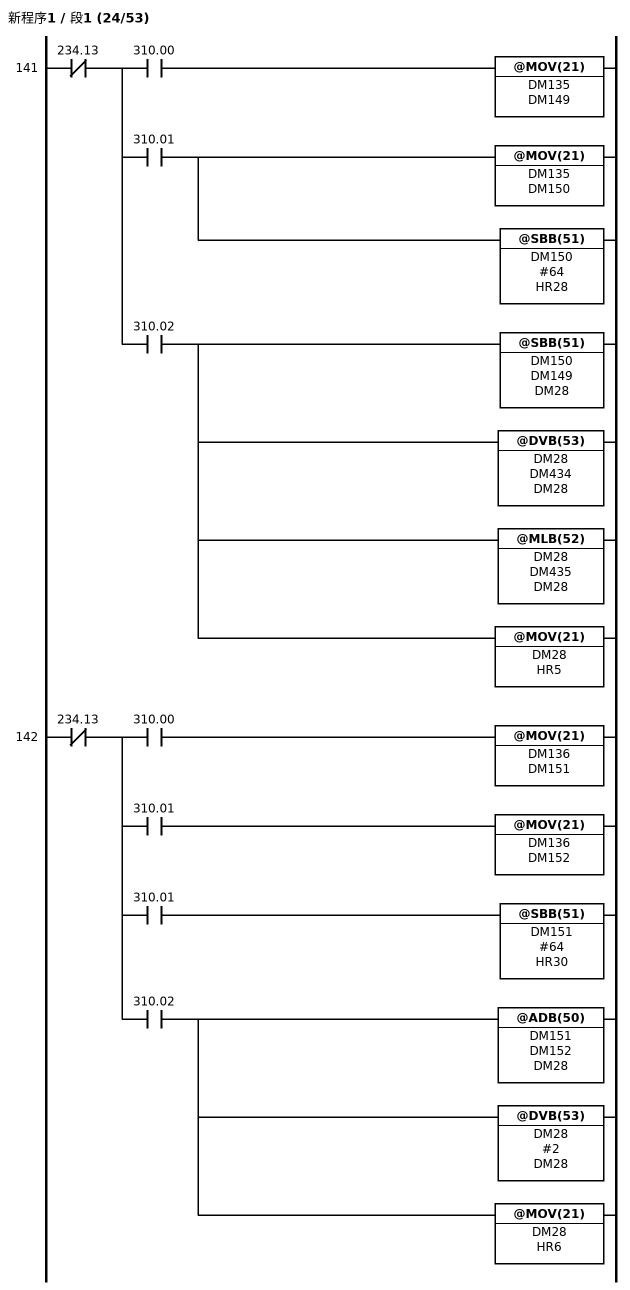
; rung 141
LDNOT 234.13
OUT TR0
AND 310.00
@MOV(21) DM135 DM149
LD TR0
AND 310.01
@MOV(21) DM135 DM150
@SBB(51) DM150 #64 HR28
LD TR0
AND 310.02
@SBB(51) DM150 DM149 DM28
@DVB(53) DM28 DM434 DM28
@MLB(52) DM28 DM435 DM28
@MOV(21) DM28 HR5
; rung 142
LDNOT 234.13
OUT TR0
AND 310.00
@MOV(21) DM136 DM151
LD TR0
AND 310.01
@MOV(21) DM136 DM152
LD TR0
AND 310.01
@SBB(51) DM151 #64 HR30
LD TR0
AND 310.02
@ADB(50) DM151 DM152 DM28
@DVB(53) DM28 #2 DM28
@MOV(21) DM28 HR6

